Yaskawa INFORM job: FRONT_WELD_0ST-2_4840_V3.JBI

/JOB
//NAME FRONT_WELD_0ST-2_4840_V3
///FOLDERNAME 02-SKRZYNIE_JOBS
//POS
///NPOS 136,136,0,25,0,0
///TOOL 0
///POSTYPE PULSE
///PULSE
C00000=1212,-39190,49707,1936,-15809,-581
C00001=-55064,-17017,13106,20113,45767,-35735
C00002=-85641,-3161,12660,31281,67420,-55579
C00003=-77611,9747,38455,32702,57795,-55547
C00004=-77611,9747,38455,32702,57795,-55547
C00005=-80481,23547,61641,37204,60115,-56891
C00006=-80479,11681,28780,33754,71138,-52780
C00007=-72683,29225,51427,31477,73582,-55335
C00008=-73419,29451,52323,31530,73467,-55649
C00009=-73173,32098,57907,31817,71820,-56064
C00010=-72655,35216,67934,32674,67821,-57152
C00011=-72655,36324,70723,32906,66918,-57452
C00012=-82806,26311,53816,38180,73291,-53604
C00013=-71695,3747,16001,30713,64750,-51022
C00014=-62587,11562,18720,19904,71589,-45519
C00015=-60535,8968,15500,19577,71351,-44837
C00016=-30585,-12603,-6778,14136,63874,-35374
C00017=13670,-17029,-10633,1297,58885,-19804
C00018=40544,-8424,-3022,-7108,61096,-10158
C00019=45161,-5697,-318,-8457,61724,-8545
C00020=46988,-9329,-5747,-8908,62911,-7987
C00021=-37830,-23193,-8618,23571,50957,-40982
C00022=11136,-28839,-12562,1025,41780,-20887
C00023=20436,-26886,-6789,-12590,38175,-10721
C00024=58488,-10629,5191,-26833,51354,2977
C00025=55110,-17412,-5825,-19778,50988,-2825
C00026=79390,11759,28162,-35512,71262,52960
C00027=82927,23281,58968,-48274,65531,63493
C00028=83399,22743,58163,-48180,65853,63532
C00029=83221,24593,61395,-48465,65231,63817
C00030=82927,34411,85507,-52086,59386,67513
C00031=76815,18630,46530,-37158,64288,54543
C00032=79390,11759,28162,-35512,71262,52960
C00033=10831,-54278,-29128,-6468,39852,-5090
C00034=-67200,-10549,24402,-3189,24913,-39001
C00035=-75122,-2194,12822,3152,39225,-43427
C00036=-77516,10189,32861,8493,33365,-45533
C00037=-90956,38945,80932,40717,38822,-71805
C00038=-88424,26013,61908,41518,40745,-70655
C00039=-82586,22930,49670,31697,49926,-67089
C00040=-80888,20314,45948,31023,49834,-66339
C00041=-77484,14865,38456,29675,49576,-64865
C00042=-77060,20165,47901,36404,58774,-63538
C00043=-73060,14132,40350,35782,57676,-62140
C00044=-77050,-3138,8526,33226,61087,-51698
C00045=-67200,-10549,24402,-3189,24913,-39001
C00046=0,-52280,40443,83103,28146,-16510
C00047=99993,-20782,22705,-13349,24734,56519
C00048=67200,-10549,24402,3189,24913,39001
C00049=75122,-2194,12822,-3152,39225,43427
C00050=74323,5203,27259,-5972,33194,43789
C00051=90148,33172,73654,-41747,37164,70694
C00052=83096,25978,54757,-26114,42930,63335
C00053=81467,18821,46286,-33706,48183,69611
C00054=80444,17239,44260,-33348,47977,69203
C00055=76924,12066,37530,-32042,47318,67771
C00056=65553,548,23705,-27852,44198,63364
C00057=76675,30944,68282,-39831,63215,59660
C00058=77050,-3138,8526,-33226,61087,51698
C00059=67200,-10549,24402,3189,24913,39001
C00060=0,-52280,40443,-83103,28146,16510
C00061=-99993,-20782,22705,13349,24734,-56519
C00062=-91125,453,39555,30378,52425,-51131
C00063=-81425,-5449,14825,37552,56592,-47667
C00064=-81425,-10835,-2515,34915,62871,-45127
C00065=-79239,4305,16082,37593,68846,-50182
C00066=-83523,16585,41906,47112,68321,-58375
C00067=-83466,26209,67230,50527,61769,-62335
C00068=-83442,29914,76031,51903,59779,-63702
C00069=-84288,15645,43522,43516,65950,-57098
C00070=-90096,4679,14083,37467,76581,-51973
C00071=-87885,29238,52923,40761,81198,69685
C00072=-84355,23847,39024,40698,83720,72224
C00073=-81800,26856,46237,41070,80563,71973
C00074=-77565,33306,56751,41640,76905,72189
C00075=-90480,18737,31939,47254,81986,71631
C00076=-94217,10634,17426,46901,86469,-59967
C00077=-81425,-10835,-2515,34915,62871,-45127
C00078=-81425,-5449,14825,37552,56592,-47667
C00079=-94290,-610,44819,32366,49686,-53459
C00080=0,-55136,17047,60468,32096,-4233
C00081=99993,-20782,22705,-13349,24734,56519
C00082=91125,453,39555,-30378,52425,51131
C00083=81425,-5449,14825,-37552,56592,47667
C00084=81425,-10835,-2515,-34915,62871,45127
C00085=79239,4305,16082,-37593,68846,50182
C00086=80765,23031,47100,-43000,73595,58456
C00087=80765,35859,79857,-46269,64609,63023
C00088=80823,37330,83115,-46640,63872,63465
C00089=85941,25971,55116,-43219,73599,60726
C00090=79256,17348,34699,-33448,76412,88212
C00091=79932,23608,50901,-39863,71219,88955
C00092=76220,30771,63034,-41386,67395,88927
C00093=86322,16060,37848,-39554,76452,89287
C00094=87424,-1569,9538,-38190,72401,52253
C00095=81425,-10835,-2515,-34915,62871,45127
C00096=92850,-11266,9233,-39092,60986,50964
C00097=28366,-40369,19479,-5635,23506,17663
C00098=-80334,-19501,31260,21216,42469,-40219
C00099=-80621,-32280,-9061,25825,59412,-41877
C00100=-80621,-37319,-22868,24573,64555,-40576
C00101=-75108,-2453,16462,35304,60348,-42510
C00102=-67175,15662,34500,25783,66040,-40361
C00103=-63819,10811,28210,25286,65654,-39198
C00104=-38821,-5630,6821,20256,64855,-32661
C00105=-39606,-22901,-1163,28356,44724,-32188
C00106=15344,-29112,-5358,-2858,33820,-6852
C00107=-15371,-20030,-486,16660,46669,-23704
C00108=-9853,-20627,-905,14451,45509,-21513
C00109=-7445,-17870,3157,22717,46629,-31388
C00110=31591,-7810,7118,6041,50959,-11062
C00111=34068,-6802,8108,5072,50869,-10082
C00112=60973,-17187,4937,-27817,44388,13718
C00113=60973,-17187,4937,-27817,44388,13718
C00114=-13287,-42463,-12044,19170,31021,-23010
C00115=-44689,-11301,43740,58858,38232,-54559
C00116=-16758,-16458,39875,62034,24713,-49593
C00117=-14258,-15900,40993,62602,23397,-49317
C00118=23190,-15776,36048,23107,10441,-22324
C00119=25491,-16071,34474,15099,11044,-17934
C00120=38205,-15598,27209,-15118,21388,-129
C00121=53765,-9366,32698,-27903,25609,9141
C00122=64054,-19541,3059,-29141,44956,15011
C00123=51466,-33957,-1499,-46586,51805,23434
C00124=44449,-8800,40981,-49870,46760,36563
C00125=21679,-14243,36560,-51489,36161,31843
C00126=19802,-15063,35701,-51447,35326,31376
C00127=-13677,-14677,25178,-29621,31481,12337
C00128=-14768,-15074,24338,-28864,31394,11719
C00129=-18871,-13754,25458,-25898,30364,9180
C00130=-35243,-10059,28499,-14440,27469,206
C00131=-36052,-9791,28742,-13797,27379,-270
C00132=-71680,-19835,10874,33863,39440,-36917
C00133=-20806,-37586,-12792,9951,42782,-18031
///LIMIT ON
C00134=29087,-45372,27330,-13325,19529,9021
C00135=0,-35121,73515,0,-2982,0
///LIMIT OFF
BC00000=801751
BC00001=853703
BC00002=856962
BC00003=856962
BC00004=856962
BC00005=856962
BC00006=873824
BC00007=873826
BC00008=873826
BC00009=873826
BC00010=873826
BC00011=873826
BC00012=873826
BC00013=873826
BC00014=873826
BC00015=873826
BC00016=873826
BC00017=873826
BC00018=873826
BC00019=873826
BC00020=919909
BC00021=919909
BC00022=919909
BC00023=919908
BC00024=919909
BC00025=873827
BC00026=873827
BC00027=873825
BC00028=873825
BC00029=873825
BC00030=873825
BC00031=873827
BC00032=873827
BC00033=869337
BC00034=845485
BC00035=874662
BC00036=874665
BC00037=874665
BC00038=874662
BC00039=874663
BC00040=874663
BC00041=874663
BC00042=874665
BC00043=874665
BC00044=874665
BC00045=845485
BC00046=774091
BC00047=774091
BC00048=845485
BC00049=874662
BC00050=874665
BC00051=874665
BC00052=874665
BC00053=874665
BC00054=874665
BC00055=874665
BC00056=874665
BC00057=874666
BC00058=874665
BC00059=845485
BC00060=774091
BC00061=774091
BC00062=811553
BC00063=857356
BC00064=876753
BC00065=876755
BC00066=876755
BC00067=876755
BC00068=876755
BC00069=876755
BC00070=877331
BC00071=876755
BC00072=890694
BC00073=890694
BC00074=890694
BC00075=890694
BC00076=890694
BC00077=876753
BC00078=857356
BC00079=811553
BC00080=811839
BC00081=774091
BC00082=811553
BC00083=857356
BC00084=876753
BC00085=876755
BC00086=876755
BC00087=876755
BC00088=876755
BC00089=876755
BC00090=876755
BC00091=876755
BC00092=876755
BC00093=876755
BC00094=876755
BC00095=876753
BC00096=857356
BC00097=788368
BC00098=802846
BC00099=822406
BC00100=860711
BC00101=860711
BC00102=860711
BC00103=860711
BC00104=860711
BC00105=906794
BC00106=906794
BC00107=860711
BC00108=860711
BC00109=860711
BC00110=860709
BC00111=860709
BC00112=860711
BC00113=853376
BC00114=860711
BC00115=860711
BC00116=860711
BC00117=860711
BC00118=860711
BC00119=860709
BC00120=860709
BC00121=860709
BC00122=860711
BC00123=860711
BC00124=860707
BC00125=860707
BC00126=860707
BC00127=860707
BC00128=860707
BC00129=860707
BC00130=860707
BC00131=860707
BC00132=860711
BC00133=857303
BC00134=744079
BC00135=636237
///POSTYPE BASE
///RECTAN
///RCONF 0,0,0,0,0,0,0,0,0,0,0,0,0,0,0,0,0,0,0,0,0,0,0,0
P00021=6.550,-0.003,-5.735,0.0000,0.0000,0.0000
P00022=5.943,-0.018,-6.388,0.0000,0.0000,0.0000
P00023=7.025,-0.019,-7.168,0.0000,0.0000,0.0000
P00024=5.926,-0.047,-4.777,0.0000,0.0000,0.0000
P00350=11.519,-0.008,1.149,0.0000,0.0000,0.0000
P00351=13.563,-0.027,-0.653,0.0000,0.0000,0.0000
P00352=13.252,-0.027,-0.827,0.0000,0.0000,0.0000
P00353=10.971,-0.082,0.776,0.0000,0.0000,0.0000
P00399=-2.449,0.031,8.825,0.0000,0.0000,0.0000
P00400=5.920,-3.503,-0.024,0.0000,0.0000,0.0000
P00401=3.430,-0.021,1.131,0.0000,0.0000,0.0000
P00402=-0.253,1.107,3.062,0.0000,0.0000,0.0000
P00403=-3.666,-0.015,5.328,0.0000,0.0000,0.0000
P00405=2.420,0.007,1.427,0.0000,0.0000,0.0000
P00406=3.513,-0.022,0.429,0.0000,0.0000,0.0000
P00415=-1.781,-1.303,3.250,0.0000,0.0000,0.0000
P00416=0.027,1.119,3.078,0.0000,0.0000,0.0000
P00420=-0.017,0.555,2.209,0.0000,0.0000,0.0000
P00421=4.378,0.044,2.315,0.0000,0.0000,0.0000
P00422=2.474,0.026,-1.450,0.0000,0.0000,0.0000
P00423=4.044,0.004,-2.619,0.0000,0.0000,0.0000
P00424=-0.387,-0.003,1.304,0.0000,0.0000,0.0000
P00425=-1.050,0.029,1.708,0.0000,0.0000,0.0000
P00426=0.002,-0.749,-0.024,0.0000,0.0000,0.0000
P00427=-1.030,-0.025,3.232,0.0000,0.0000,0.0000
//INST
///DATE 2025/06/04 08:20
///ATTR SC,RW
///GROUP1 RB1,BS1
NOP
'**********************
'**********************
'POCZATEK SPAWANIA PRZOD
'**********************
'**********************
MOVJ C00000 BC00000 VJ=60.00
MOVL C00001 BC00001 V=416.7
MOVJ C00002 BC00002 VJ=10.00
MOVJ C00003 BC00003 VJ=10.00
MOVL C00004 BC00004 V=150.0
MOVL C00005 BC00005 V=150.0
'**********************
'W41A SIDE
'**********************
MOVL C00006 BC00006 V=250.0
SFTON P0402
MOVL C00007 BC00007 V=66.7 PL=0
REFP 1 C00008 BC00008
REFP 2 C00009 BC00009
MACRO1 MJ#(0) ARGF14
ARCON
WVON WEV#(5)
MOVL C00010 BC00010 V=9.2
MOVL C00011 BC00011 V=9.2
ARCOF
WVOF
SFTOF
MOVL C00012 BC00012 V=166.7
'**********************
'W41A FRONT
'**********************
MOVL C00013 BC00013 V=250.0
SFTON P0350
MOVL C00014 BC00014 V=66.7 PL=0
MACRO1 MJ#(0) ARGF21
ARCON
COMM WVON WEV#(2)
MOVL C00015 BC00015 V=6.7
SFTON P0351
MOVL C00016 BC00016 V=6.7
SFTON P0352
MOVL C00017 BC00017 V=6.7
SFTON P0353
MOVL C00018 BC00018 V=6.7
MOVL C00019 BC00019 V=6.7
SFTOF
ARCOF
WVOF
COMM MOVL C00020 BC00020 V=166.7
COMM MOVL C00021 BC00021 V=166.7
COMM '**********************
COMM 'W41B FRONT
COMM '**********************
COMM MOVL C00022 BC00022 V=250.0
COMM SFTON P0352
COMM MOVL C00023 BC00023 V=66.7 PL=0
COMM SFTOF
COMM MACRO1 MJ#(0) ARGF21
COMM ARCON
COMM WVON WEV#(2)
COMM SFTON P0353
COMM MOVL C00024 BC00024 V=8.3
COMM SFTOF
COMM ARCOF
COMM WVOF
MOVL C00025 BC00025 V=166.7
MOVL C00026 BC00026 V=100.0
'**********************
'W41A SIDE
'**********************
SFTON P0400
MOVL C00027 BC00027 V=66.7 PL=0
MACRO1 MJ#(0) ARGF21
REFP 1 C00028 BC00028
REFP 2 C00029 BC00029
ARCON
WVON WEV#(5)
MOVL C00030 BC00030 V=8.3
ARCOF
WVOF
SFTOF
MOVL C00031 BC00031 V=83.3
MOVL C00032 BC00032 V=166.7
MOVL C00033 BC00033 V=333.3
MOVJ C00034 BC00034 VJ=20.00
MOVJ C00035 BC00035 VJ=20.00
'**********************
'W42A.1
'**********************
'POPRAWIC
MOVL C00036 BC00036 V=500.0
SFTON P0403
MOVL C00037 BC00037 V=66.7 PL=0
MACRO1 MJ#(0) ARGF9
ARCON
MOVL C00038 BC00038 V=9.2
SFTON P0416
MOVL C00039 BC00039 V=9.2
MOVL C00040 BC00040 V=9.2
MOVL C00041 BC00041 V=9.2
SFTON P0421
MOVL C00042 BC00042 V=9.2
SFTON P0402
MOVL C00043 BC00043 V=9.2
ARCOF
MOVL C00044 BC00044 V=500.0
SFTOF
MOVJ C00045 BC00045 VJ=15.00
'W42B.1
MOVJ C00046 BC00046 VJ=30.00
MOVJ C00047 BC00047 VJ=30.00
MOVJ C00048 BC00048 VJ=30.00
MOVJ C00049 BC00049 VJ=30.00
'**********************
'W42B.1
'**********************
MOVL C00050 BC00050 V=500.0
SFTON P0399
MOVL C00051 BC00051 V=166.7 PL=0
MACRO1 MJ#(0) ARGF9
ARCON
MOVL C00052 BC00052 V=8.3
SFTON P0415
MOVL C00053 BC00053 V=9.2
MOVL C00054 BC00054 V=9.2
MOVL C00055 BC00055 V=9.2
SFTON P0427
MOVL C00056 BC00056 V=9.2
SFTON P0400
MOVL C00057 BC00057 V=9.2
ARCOF
MOVL C00058 BC00058 V=83.3 PL=0
SFTOF
MOVJ C00059 BC00059 VJ=25.00
'W42A.2
MOVJ C00060 BC00060 VJ=40.00
MOVJ C00061 BC00061 VJ=30.00
MOVJ C00062 BC00062 VJ=30.00
MOVJ C00063 BC00063 VJ=30.00
MOVJ C00064 BC00064 VJ=30.00
'**********************
'W42A.2
'**********************
MOVL C00065 BC00065 V=500.0
SFTON P0420
MOVL C00066 BC00066 V=166.7 PL=0
SFTOF
MACRO1 MJ#(0) ARGF9
ARCON
WVON WEV#(6)
MOVL C00067 BC00067 V=9.2
SFTON P0402
MOVL C00068 BC00068 V=9.2
ARCOF
WVOF
MOVL C00069 BC00069 V=166.7
MOVJ C00070 BC00070 VJ=20.00
MOVJ C00071 BC00071 VJ=20.00
MOVL C00072 BC00072 V=250.0
MOVL C00073 BC00073 V=166.7
ARCON
MOVL C00074 BC00074 V=10.8
ARCOF
MOVL C00075 BC00075 V=166.7
MOVJ C00076 BC00076 VJ=20.00
SFTOF
MOVJ C00077 BC00077 VJ=30.00
MOVJ C00078 BC00078 VJ=30.00
MOVJ C00079 BC00079 VJ=30.00
'W42B.2
MOVJ C00080 BC00080 VJ=30.00
MOVJ C00081 BC00081 VJ=30.00
MOVJ C00082 BC00082 VJ=30.00
MOVJ C00083 BC00083 VJ=30.00
MOVJ C00084 BC00084 VJ=30.00
'**********************
'W42B.2
'**********************
MOVL C00085 BC00085 V=500.0
SFTON P0426
MOVL C00086 BC00086 V=166.7 PL=0
SFTOF
MACRO1 MJ#(0) ARGF9
ARCON
WVON WEV#(6)
MOVL C00087 BC00087 V=9.2
SFTON P0400
MOVL C00088 BC00088 V=9.2
ARCOF
WVOF
SFTOF
MOVL C00089 BC00089 V=166.7
MOVJ C00090 BC00090 VJ=10.00
SFTON P0400
MOVL C00091 BC00091 V=166.7
ARCON
MOVL C00092 BC00092 V=10.8
ARCOF
MOVL C00093 BC00093 V=250.0
MOVL C00094 BC00094 V=500.0
SFTOF
MOVJ C00095 BC00095 VJ=20.00
MOVJ C00096 BC00096 VJ=30.00
'W42A.3
MOVJ C00097 BC00097 VJ=20.00
MOVJ C00098 BC00098 VJ=20.00
MOVJ C00099 BC00099 VJ=30.00
MOVJ C00100 BC00100 VJ=30.00
'**********************
'W42A.3
'**********************
MOVL C00101 BC00101 V=500.0
SFTON P0021
MOVL C00102 BC00102 V=166.7 PL=0
MACRO1 MJ#(0) ARGF9
ARCON
MOVL C00103 BC00103 V=8.3
COMM WVON WEV#(2)
SFTON P0022
MOVL C00104 BC00104 V=8.3
COMM ARCOF
COMM WVOF
COMM MOVL C00105 BC00105 V=500.0
COMM SFTOF
COMM '**********************
COMM 'W42B.3
COMM '**********************
COMM MOVL C00106 BC00106 V=500.0
SFTON P0023
MOVL C00107 BC00107 V=8.3
WVON WEV#(2)
MOVL C00108 BC00108 V=6.7
WVOF
MOVL C00109 BC00109 V=8.3
SFTON P0024
MOVL C00110 BC00110 V=8.3
MOVL C00111 BC00111 V=8.3
ARCOF
WVOF
MOVL C00112 BC00112 V=500.0
SFTOF
MOVJ C00113 BC00113 VJ=20.00
'**********************
'GORA L
'**********************
MOVL C00114 BC00114 V=500.0
SFTON P0401
MOVL C00115 BC00115 V=166.7 PL=0
MACRO1 MJ#(0) ARGF9
ARCON
MOVL C00116 BC00116 V=11.7
SFTON P0424
MOVL C00117 BC00117 V=11.7
SFTON P0425
MOVL C00118 BC00118 V=11.7
SFTON P0406
MOVL C00119 BC00119 V=11.7
MOVL C00120 BC00120 V=11.7
MOVL C00121 BC00121 V=11.7
ARCOF
MOVL C00122 BC00122 V=500.0
SFTOF
'**********************
'GORA P
'**********************
MOVL C00123 BC00123 V=166.7
SFTON P0401
MOVL C00124 BC00124 V=166.7 PL=0
ARCON
MOVL C00125 BC00125 V=11.7
SFTON P0423
MOVL C00126 BC00126 V=11.7
SFTON P0422
MOVL C00127 BC00127 V=11.7
MOVL C00128 BC00128 V=11.7
SFTON P0405
MOVL C00129 BC00129 V=11.7
MOVL C00130 BC00130 V=11.7
MOVL C00131 BC00131 V=11.7
ARCOF
MOVL C00132 BC00132 V=500.0
SFTOF
MOVJ C00133 BC00133 VJ=20.00
MOVJ C00134 BC00134 VJ=30.00
MOVJ C00135 BC00135 VJ=30.00
'KONIEC SPAWANIA FRONTU
END
